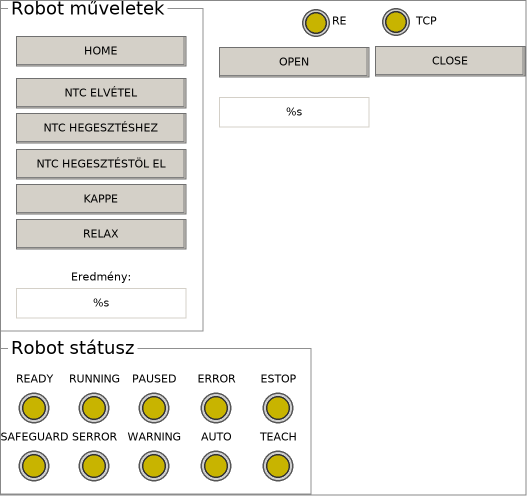
VISUALIZATION TempRobot  // 527x496
    Button (219,47 150x30), "OPEN", invisible if: RobotProcess.iState>0, input disabled if: RobotProcess.iState>0
        OnMouseClick: execute { RobotProcess.iState:=1; }
    Button (375,46 150x30), "CLOSE", invisible if: RobotProcess.iState=0, input disabled if: RobotProcess.iState=0
        OnMouseClick: execute { RobotProcess.iState:=200; }
    Lamp1 (298,7 36x32), variable: ROBOTREMOTE.bRobotCommOpen, style: Lamp-Lamp1-Yellow
    Label (311,6 57x30), "RE"
    Label (398,6 57x30), "TCP"
    Lamp1 (378,6 36x32), variable: ROBOTCOMMAND.bRobotCommOpen, style: Lamp-Lamp1-Yellow
    GroupBox (0,340 311x154), "Robot státusz"
        Lamp1 (16,50 36x36), variable: RobotProcess.baStatus[10], invisible if: ROBOTREMOTE.bRobotCommOpen=FALSE, style: Lamp-Lamp1-Yellow
        Label (6,24 57x30), "READY", invisible if: ROBOTREMOTE.bRobotCommOpen=FALSE
        Lamp1 (76,50 36x36), variable: RobotProcess.baStatus[9], invisible if: ROBOTREMOTE.bRobotCommOpen=FALSE, style: Lamp-Lamp1-Yellow
        Label (66,24 57x30), "RUNNING", invisible if: ROBOTREMOTE.bRobotCommOpen=FALSE
        Lamp1 (136,50 36x36), variable: RobotProcess.baStatus[8], invisible if: ROBOTREMOTE.bRobotCommOpen=FALSE, style: Lamp-Lamp1-Yellow
        Label (126,24 57x30), "PAUSED", invisible if: ROBOTREMOTE.bRobotCommOpen=FALSE
        Lamp1 (198,50 36x36), variable: RobotProcess.baStatus[7], invisible if: ROBOTREMOTE.bRobotCommOpen=FALSE, style: Lamp-Lamp1-Yellow
        Label (188,24 57x30), "ERROR", invisible if: ROBOTREMOTE.bRobotCommOpen=FALSE
        Lamp1 (260,50 36x36), variable: RobotProcess.baStatus[6], invisible if: ROBOTREMOTE.bRobotCommOpen=FALSE, style: Lamp-Lamp1-Yellow
        Label (250,24 57x30), "ESTOP", invisible if: ROBOTREMOTE.bRobotCommOpen=FALSE
        Lamp1 (16,108 36x36), variable: RobotProcess.baStatus[5], invisible if: ROBOTREMOTE.bRobotCommOpen=FALSE, style: Lamp-Lamp1-Yellow
        Label (6,82 57x30), "SAFEGUARD", invisible if: ROBOTREMOTE.bRobotCommOpen=FALSE
        Lamp1 (76,108 36x36), variable: RobotProcess.baStatus[4], invisible if: ROBOTREMOTE.bRobotCommOpen=FALSE, style: Lamp-Lamp1-Yellow
        Label (66,82 57x30), "SERROR", invisible if: ROBOTREMOTE.bRobotCommOpen=FALSE
        Lamp1 (136,108 36x36), variable: RobotProcess.baStatus[3], invisible if: ROBOTREMOTE.bRobotCommOpen=FALSE, style: Lamp-Lamp1-Yellow
        Label (126,82 57x30), "WARNING", invisible if: ROBOTREMOTE.bRobotCommOpen=FALSE
        Lamp1 (198,108 36x36), variable: RobotProcess.baStatus[2], invisible if: ROBOTREMOTE.bRobotCommOpen=FALSE, style: Lamp-Lamp1-Yellow
        Label (188,82 57x30), "AUTO", invisible if: ROBOTREMOTE.bRobotCommOpen=FALSE
        Lamp1 (260,108 36x36), variable: RobotProcess.baStatus[1], invisible if: ROBOTREMOTE.bRobotCommOpen=FALSE, style: Lamp-Lamp1-Yellow
        Label (250,82 57x30), "TEACH", invisible if: ROBOTREMOTE.bRobotCommOpen=FALSE
    GroupBox (0,0 203x331), "Robot műveletek"
        Button (16,78 170x30), "NTC ELVÉTEL", invisible if: RobotProcess.iState=0, input disabled if: RobotProcess.iState=0
            OnMouseClick: execute { RobotProcess.s_InRobotTCPCommand := 'NTCHEZ'; }
        Button (16,113 170x30), "NTC HEGESZTÉSHEZ", invisible if: RobotProcess.iState=0, input disabled if: RobotProcess.iState=0
            OnMouseClick: execute { RobotProcess.s_InRobotTCPCommand := 'NTCHEG'; }
        Button (16,149 170x30), "NTC HEGESZTÉSTÖL EL", invisible if: RobotProcess.iState=0, input disabled if: RobotProcess.iState=0
            OnMouseClick: execute { RobotProcess.s_InRobotTCPCommand := 'NTCHEGTOL'; }
        Button (16,184 170x30), "KAPPE", invisible if: RobotProcess.iState=0, input disabled if: RobotProcess.iState=0
            OnMouseClick: execute { RobotProcess.s_InRobotTCPCommand := 'KAPPE'; }
        Button (16,219 170x30), "RELAX", invisible if: RobotProcess.iState=0, input disabled if: RobotProcess.iState=0
            OnMouseClick: execute { RobotProcess.s_InRobotTCPCommand := 'RELAX'; }
        Button (16,36 170x30), "HOME", invisible if: RobotProcess.iState=0, input disabled if: RobotProcess.iState=0
            OnMouseClick: execute { RobotProcess.s_InRobotTCPCommand := 'HOME'; }
        Label (56,262 90x30), "Eredmény:"
        Textfield (16,288 170x30), "%s", text variable: ROBOTCOMMAND.sRobotResult, input disabled if: TRUE
    Textfield (219,97 150x30), "%s", text variable: RobotProcess.iState, input disabled if: TRUE
END_VISUALIZATION

(* stored: Version 1.1.0.1, ProductVersion 3.1.4024.11
   Visu TempRobot: Id {afc3fa60-523e-45c8-a515-595c085d90eb} *)
